{attribute 'linkalways'} 
{attribute 'no_explicit_call' := 'This FB is a CLASS and must be accessed using methods or properties'}
{attribute 'enable_dynamic_creation'}
FUNCTION_BLOCK FINAL LE_LWORD EXTENDS Node
VAR
	in1 : _LWORD(0);
	in2 : _LWORD(0);
	out : _BOOL(FALSE);
END_VAR

METHOD PUBLIC Clone : I_Node
VAR
	pNode : POINTER TO LE_LWORD;
END_VAR
pNode := __NEW(LE_LWORD);
Clone := pNode^;
END_METHOD

METHOD FB_init : BOOL
VAR_INPUT
	bInitRetains : BOOL; // if TRUE, the retain variables are initialized (warm start / cold start)
	bInCopyCode : BOOL;  // if TRUE, the instance afterwards gets moved into the copy code (online change)
END_VAR
AddInput('in1',THIS^.in1);
AddInput('in2',THIS^.in2);
AddOutput('out', THIS^.out);
END_METHOD

METHOD PROTECTED OnExecute
VAR
END_VAR
out.Value := in1.Value <= in2.Value;
END_METHOD

END_FUNCTION_BLOCK

(* stored: Version 1.1.0.1, ProductVersion 3.1.4024.15
   POU LE_LWORD: Id {204de4c2-6127-48f7-85a2-5067513d9d55}, SpecialFunc None
   Folder Constructor: Id {8f4d9a9d-5c92-4df4-8cbe-a14630d75e45}
   Method Clone: Id {a3185fee-1692-413d-8fd1-71190eb0f7c5}
   Method FB_init: Id {a0a8dd71-e42e-471e-90e7-38ee455ebbde}
   Method OnExecute: Id {bffcf8ab-e1e2-44ee-b420-134dce662080} *)
